FUNCTION_BLOCK Component_Mockup EXTENDS Component
VAR
END_VAR

END_FUNCTION_BLOCK

(* stored: Version 1.1.0.1, ProductVersion 3.1.4026.18
   POU Component_Mockup: Id {9389c20d-c061-49ef-9b74-f44986cbfc34}, SpecialFunc None *)
